{attribute 'qualified_only'}
{attribute 'strict'}
TYPE StartType :
(
	Absolute := 1,
	Relative := 2,
	VeloPositive := 3,
	VeloNegative := 4,
	Calibrate := 24576 
);
END_TYPE

(* stored: Version 1.1.0.1, ProductVersion 3.1.4024.11
   DUT StartType: Id {ee0510c6-31de-4f02-b260-45f4bb61e15b} *)
